GLOBALCONSTANTS DefaultPool_PWM12_Numeric (* Numeric object pool constants (ID, Scale, Offset, Decimals) *)
  PACKAGE Uebungen::const::UT::PWM12;
  VAR_GLOBAL CONSTANT
    InputNumber_PWM_Q01_N : logiBUS::utils::conversion::phys::NumericObjectPool_S := (u16ObjId := 9000, r32Scale := 0.0015560939, i32Offset := 0, u8Decimals := 3);
    InputNumber_PWM_Q02_N : logiBUS::utils::conversion::phys::NumericObjectPool_S := (u16ObjId := 9001, r32Scale := 0.0015560939, i32Offset := 0, u8Decimals := 3);
    InputNumber_PWM_Q03_N : logiBUS::utils::conversion::phys::NumericObjectPool_S := (u16ObjId := 9002, r32Scale := 0.0015560939, i32Offset := 0, u8Decimals := 3);
    InputNumber_PWM_Q04_N : logiBUS::utils::conversion::phys::NumericObjectPool_S := (u16ObjId := 9003, r32Scale := 0.0015560939, i32Offset := 0, u8Decimals := 3);
    InputNumber_PWM_Q05_N : logiBUS::utils::conversion::phys::NumericObjectPool_S := (u16ObjId := 9004, r32Scale := 0.0015560939, i32Offset := 0, u8Decimals := 3);
    InputNumber_PWM_Q06_N : logiBUS::utils::conversion::phys::NumericObjectPool_S := (u16ObjId := 9005, r32Scale := 0.0015560939, i32Offset := 0, u8Decimals := 3);
    InputNumber_PWM_Q07_N : logiBUS::utils::conversion::phys::NumericObjectPool_S := (u16ObjId := 9006, r32Scale := 0.0015560939, i32Offset := 0, u8Decimals := 3);
    InputNumber_PWM_Q08_N : logiBUS::utils::conversion::phys::NumericObjectPool_S := (u16ObjId := 9007, r32Scale := 0.0015560939, i32Offset := 0, u8Decimals := 3);
    InputNumber_PWM_Q09_N : logiBUS::utils::conversion::phys::NumericObjectPool_S := (u16ObjId := 9008, r32Scale := 0.0015560939, i32Offset := 0, u8Decimals := 3);
    InputNumber_PWM_Q10_N : logiBUS::utils::conversion::phys::NumericObjectPool_S := (u16ObjId := 9009, r32Scale := 0.0015560939, i32Offset := 0, u8Decimals := 3);
    InputNumber_PWM_Q11_N : logiBUS::utils::conversion::phys::NumericObjectPool_S := (u16ObjId := 9010, r32Scale := 0.0015560939, i32Offset := 0, u8Decimals := 3);
    InputNumber_PWM_Q12_N : logiBUS::utils::conversion::phys::NumericObjectPool_S := (u16ObjId := 9011, r32Scale := 0.0015560939, i32Offset := 0, u8Decimals := 3);
    InputNumberRaw_PWM_Q01_N : logiBUS::utils::conversion::phys::NumericObjectPool_S := (u16ObjId := 9012, r32Scale := 1.0, i32Offset := 0, u8Decimals := 0);
    InputNumberRaw_PWM_Q02_N : logiBUS::utils::conversion::phys::NumericObjectPool_S := (u16ObjId := 9013, r32Scale := 1.0, i32Offset := 0, u8Decimals := 0);
    InputNumberRaw_PWM_Q03_N : logiBUS::utils::conversion::phys::NumericObjectPool_S := (u16ObjId := 9014, r32Scale := 1.0, i32Offset := 0, u8Decimals := 0);
    InputNumberRaw_PWM_Q04_N : logiBUS::utils::conversion::phys::NumericObjectPool_S := (u16ObjId := 9015, r32Scale := 1.0, i32Offset := 0, u8Decimals := 0);
    InputNumberRaw_PWM_Q05_N : logiBUS::utils::conversion::phys::NumericObjectPool_S := (u16ObjId := 9016, r32Scale := 1.0, i32Offset := 0, u8Decimals := 0);
    InputNumberRaw_PWM_Q06_N : logiBUS::utils::conversion::phys::NumericObjectPool_S := (u16ObjId := 9017, r32Scale := 1.0, i32Offset := 0, u8Decimals := 0);
    InputNumberRaw_PWM_Q07_N : logiBUS::utils::conversion::phys::NumericObjectPool_S := (u16ObjId := 9018, r32Scale := 1.0, i32Offset := 0, u8Decimals := 0);
    InputNumberRaw_PWM_Q08_N : logiBUS::utils::conversion::phys::NumericObjectPool_S := (u16ObjId := 9019, r32Scale := 1.0, i32Offset := 0, u8Decimals := 0);
    InputNumberRaw_PWM_Q09_N : logiBUS::utils::conversion::phys::NumericObjectPool_S := (u16ObjId := 9020, r32Scale := 1.0, i32Offset := 0, u8Decimals := 0);
    InputNumberRaw_PWM_Q10_N : logiBUS::utils::conversion::phys::NumericObjectPool_S := (u16ObjId := 9021, r32Scale := 1.0, i32Offset := 0, u8Decimals := 0);
    InputNumberRaw_PWM_Q11_N : logiBUS::utils::conversion::phys::NumericObjectPool_S := (u16ObjId := 9022, r32Scale := 1.0, i32Offset := 0, u8Decimals := 0);
    InputNumberRaw_PWM_Q12_N : logiBUS::utils::conversion::phys::NumericObjectPool_S := (u16ObjId := 9023, r32Scale := 1.0, i32Offset := 0, u8Decimals := 0);
    OutputNumber_c1_N : logiBUS::utils::conversion::phys::NumericObjectPool_S := (u16ObjId := 12001, r32Scale := 1.0, i32Offset := 0, u8Decimals := 0);
    OutputNumber_c2_N : logiBUS::utils::conversion::phys::NumericObjectPool_S := (u16ObjId := 12013, r32Scale := 1.0, i32Offset := 0, u8Decimals := 0);
    OutputNumber_c3_N : logiBUS::utils::conversion::phys::NumericObjectPool_S := (u16ObjId := 12014, r32Scale := 1.0, i32Offset := 0, u8Decimals := 0);
    OutputNumber_c4_N : logiBUS::utils::conversion::phys::NumericObjectPool_S := (u16ObjId := 12015, r32Scale := 1.0, i32Offset := 0, u8Decimals := 0);
    OutputNumber_c5_N : logiBUS::utils::conversion::phys::NumericObjectPool_S := (u16ObjId := 12016, r32Scale := 1.0, i32Offset := 0, u8Decimals := 0);
    OutputNumber_c6_N : logiBUS::utils::conversion::phys::NumericObjectPool_S := (u16ObjId := 12017, r32Scale := 1.0, i32Offset := 0, u8Decimals := 0);
    OutputNumber_c7_N : logiBUS::utils::conversion::phys::NumericObjectPool_S := (u16ObjId := 12018, r32Scale := 1.0, i32Offset := 0, u8Decimals := 0);
    OutputNumber_c8_N : logiBUS::utils::conversion::phys::NumericObjectPool_S := (u16ObjId := 12019, r32Scale := 1.0, i32Offset := 0, u8Decimals := 0);
    OutputNumber_Tick_N : logiBUS::utils::conversion::phys::NumericObjectPool_S := (u16ObjId := 12020, r32Scale := 1.0, i32Offset := 0, u8Decimals := 0);
    NumberVariable_PWM_Q01_N : logiBUS::utils::conversion::phys::NumericObjectPool_S := (u16ObjId := 21000, r32Scale := 0.0015560939, i32Offset := 0, u8Decimals := 3);
    NumberVariable_PWM_Q02_N : logiBUS::utils::conversion::phys::NumericObjectPool_S := (u16ObjId := 21001, r32Scale := 0.0015560939, i32Offset := 0, u8Decimals := 3);
    NumberVariable_PWM_Q03_N : logiBUS::utils::conversion::phys::NumericObjectPool_S := (u16ObjId := 21002, r32Scale := 0.0015560939, i32Offset := 0, u8Decimals := 3);
    NumberVariable_PWM_Q04_N : logiBUS::utils::conversion::phys::NumericObjectPool_S := (u16ObjId := 21003, r32Scale := 0.0015560939, i32Offset := 0, u8Decimals := 3);
    NumberVariable_PWM_Q05_N : logiBUS::utils::conversion::phys::NumericObjectPool_S := (u16ObjId := 21004, r32Scale := 0.0015560939, i32Offset := 0, u8Decimals := 3);
    NumberVariable_PWM_Q06_N : logiBUS::utils::conversion::phys::NumericObjectPool_S := (u16ObjId := 21005, r32Scale := 0.0015560939, i32Offset := 0, u8Decimals := 3);
    NumberVariable_PWM_Q07_N : logiBUS::utils::conversion::phys::NumericObjectPool_S := (u16ObjId := 21006, r32Scale := 0.0015560939, i32Offset := 0, u8Decimals := 3);
    NumberVariable_PWM_Q08_N : logiBUS::utils::conversion::phys::NumericObjectPool_S := (u16ObjId := 21007, r32Scale := 0.0015560939, i32Offset := 0, u8Decimals := 3);
    NumberVariable_PWM_Q09_N : logiBUS::utils::conversion::phys::NumericObjectPool_S := (u16ObjId := 21008, r32Scale := 0.0015560939, i32Offset := 0, u8Decimals := 3);
    NumberVariable_PWM_Q10_N : logiBUS::utils::conversion::phys::NumericObjectPool_S := (u16ObjId := 21009, r32Scale := 0.0015560939, i32Offset := 0, u8Decimals := 3);
    NumberVariable_PWM_Q11_N : logiBUS::utils::conversion::phys::NumericObjectPool_S := (u16ObjId := 21010, r32Scale := 0.0015560939, i32Offset := 0, u8Decimals := 3);
    NumberVariable_PWM_Q12_N : logiBUS::utils::conversion::phys::NumericObjectPool_S := (u16ObjId := 21011, r32Scale := 0.0015560939, i32Offset := 0, u8Decimals := 3);
  END_VAR
END_GLOBALCONSTANTS
(* other elements stored in the file *)
(* ACHTUNG: 'NumberVariable_PWM_Q01' wird von mehreren Widgets mit unterschiedlicher Skalierung gebunden - 'InputNumber_PWM_Q01' (scale=0.0015560939 offset=0 decimals=3) vs. 'InputNumberRaw_PWM_Q01' (scale=1.0 offset=0 decimals=0). Es gilt die Skalierung mit dem kleinsten |Scale|, alle Widgets muessen dieselbe Skalierung haben. *)
(* ACHTUNG: 'NumberVariable_PWM_Q02' wird von mehreren Widgets mit unterschiedlicher Skalierung gebunden - 'InputNumber_PWM_Q02' (scale=0.0015560939 offset=0 decimals=3) vs. 'InputNumberRaw_PWM_Q02' (scale=1.0 offset=0 decimals=0). Es gilt die Skalierung mit dem kleinsten |Scale|, alle Widgets muessen dieselbe Skalierung haben. *)
(* ACHTUNG: 'NumberVariable_PWM_Q03' wird von mehreren Widgets mit unterschiedlicher Skalierung gebunden - 'InputNumber_PWM_Q03' (scale=0.0015560939 offset=0 decimals=3) vs. 'InputNumberRaw_PWM_Q03' (scale=1.0 offset=0 decimals=0). Es gilt die Skalierung mit dem kleinsten |Scale|, alle Widgets muessen dieselbe Skalierung haben. *)
(* ACHTUNG: 'NumberVariable_PWM_Q04' wird von mehreren Widgets mit unterschiedlicher Skalierung gebunden - 'InputNumber_PWM_Q04' (scale=0.0015560939 offset=0 decimals=3) vs. 'InputNumberRaw_PWM_Q04' (scale=1.0 offset=0 decimals=0). Es gilt die Skalierung mit dem kleinsten |Scale|, alle Widgets muessen dieselbe Skalierung haben. *)
(* ACHTUNG: 'NumberVariable_PWM_Q05' wird von mehreren Widgets mit unterschiedlicher Skalierung gebunden - 'InputNumber_PWM_Q05' (scale=0.0015560939 offset=0 decimals=3) vs. 'InputNumberRaw_PWM_Q05' (scale=1.0 offset=0 decimals=0). Es gilt die Skalierung mit dem kleinsten |Scale|, alle Widgets muessen dieselbe Skalierung haben. *)
(* ACHTUNG: 'NumberVariable_PWM_Q06' wird von mehreren Widgets mit unterschiedlicher Skalierung gebunden - 'InputNumber_PWM_Q06' (scale=0.0015560939 offset=0 decimals=3) vs. 'InputNumberRaw_PWM_Q06' (scale=1.0 offset=0 decimals=0). Es gilt die Skalierung mit dem kleinsten |Scale|, alle Widgets muessen dieselbe Skalierung haben. *)
(* ACHTUNG: 'NumberVariable_PWM_Q07' wird von mehreren Widgets mit unterschiedlicher Skalierung gebunden - 'InputNumber_PWM_Q07' (scale=0.0015560939 offset=0 decimals=3) vs. 'InputNumberRaw_PWM_Q07' (scale=1.0 offset=0 decimals=0). Es gilt die Skalierung mit dem kleinsten |Scale|, alle Widgets muessen dieselbe Skalierung haben. *)
(* ACHTUNG: 'NumberVariable_PWM_Q08' wird von mehreren Widgets mit unterschiedlicher Skalierung gebunden - 'InputNumber_PWM_Q08' (scale=0.0015560939 offset=0 decimals=3) vs. 'InputNumberRaw_PWM_Q08' (scale=1.0 offset=0 decimals=0). Es gilt die Skalierung mit dem kleinsten |Scale|, alle Widgets muessen dieselbe Skalierung haben. *)
(* ACHTUNG: 'NumberVariable_PWM_Q09' wird von mehreren Widgets mit unterschiedlicher Skalierung gebunden - 'InputNumber_PWM_Q09' (scale=0.0015560939 offset=0 decimals=3) vs. 'InputNumberRaw_PWM_Q09' (scale=1.0 offset=0 decimals=0). Es gilt die Skalierung mit dem kleinsten |Scale|, alle Widgets muessen dieselbe Skalierung haben. *)
(* ACHTUNG: 'NumberVariable_PWM_Q10' wird von mehreren Widgets mit unterschiedlicher Skalierung gebunden - 'InputNumber_PWM_Q10' (scale=0.0015560939 offset=0 decimals=3) vs. 'InputNumberRaw_PWM_Q10' (scale=1.0 offset=0 decimals=0). Es gilt die Skalierung mit dem kleinsten |Scale|, alle Widgets muessen dieselbe Skalierung haben. *)
(* ACHTUNG: 'NumberVariable_PWM_Q11' wird von mehreren Widgets mit unterschiedlicher Skalierung gebunden - 'InputNumber_PWM_Q11' (scale=0.0015560939 offset=0 decimals=3) vs. 'InputNumberRaw_PWM_Q11' (scale=1.0 offset=0 decimals=0). Es gilt die Skalierung mit dem kleinsten |Scale|, alle Widgets muessen dieselbe Skalierung haben. *)
(* ACHTUNG: 'NumberVariable_PWM_Q12' wird von mehreren Widgets mit unterschiedlicher Skalierung gebunden - 'InputNumber_PWM_Q12' (scale=0.0015560939 offset=0 decimals=3) vs. 'InputNumberRaw_PWM_Q12' (scale=1.0 offset=0 decimals=0). Es gilt die Skalierung mit dem kleinsten |Scale|, alle Widgets muessen dieselbe Skalierung haben. *)
